Universal Robots PolyScope program: network_test.urp

Program network_test (installation=default directory=/programs/usbdisk_1/TVT19SPL createdIn=5.11.5.1010327 lastSavedIn=5.11.5.1010327 robotSerialNumber=20195600355)
Calibrated DH parameters: a=[0.000056, -0.161146, -0.252643, 0.000052, -0.000071, 0]; d=[0.181245, -342.672485, 975.135632, -632.288651, 0.119957, 0.115765]; alpha=[1.571164, 0.001314, -0.000405, 1.570615, -1.570559, 0]; deltaTheta=[0, -1.227166, 0.434415, 0.792759, -0.000001, 0]
BeforeStart
  pcip := "10.42.0.1"
  connection1 := False
  Loop While (checkContinuously=false) expression=not connection1
    connection1 := socket_open(pcip,1201)
Robot Program (runOnlyOnce=false)
  Script: socket_send_string("Test packet")
  recieve_srv := socket_read_string(timeout=0)
  If recieve_srv≟"1"
    MoveJ speed 60 deg/s, acceleration 80 deg/s^2 (useActiveTCP=true) feature=Base
      Waypoint Waypoint_1: TCP in base x=-26.202 y=-417.811 z=164.679 mm, rx=-2.4767 ry=-0.1631 rz=-0.0534 rad; joints [70.184, -71.361, 101.909, -84.408, -102.174, 156.626] deg; TCP offset x=0 y=0 z=158.01 mm, rx=0 ry=0 rz=0 rad
  ElseIf recieve_srv≟"2"
    MoveJ speed 60 deg/s, acceleration 80 deg/s^2 (useActiveTCP=true) feature=Base
      Waypoint Waypoint_2: TCP in base x=-22.57 y=-506.108 z=514.303 mm, rx=-3.0137 ry=-0.2292 rz=0.0658 rad; joints [70.208, -83.067, 60.073, -61.802, -95.097, 151.742] deg
